FUNCTION_BLOCK INTEGRAL (* determines approximately the integral over time. *)
  (* Standard: 61499-1; Description: Copyright (c) 2024 HR Agrartechnik GmbH This program and the accompanying materials are made available under the terms of the Eclipse Public License 2.0 which is available at https://www.eclipse.org/legal/epl-2.0/ SPDX-License-Identifier: EPL-2.0 This Block was inspired by https://content.helpme-codesys.com/en/libs/Util/Current/Mathematical-Functions/INTEGRAL.html *)
  (* Version 1.0, 2024-10-18, Franz Höpfinger, HR Agrartechnik GmbH, initial Version *)
  PACKAGE utils::math;
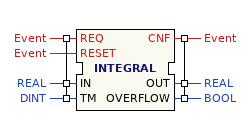
  EVENT_INPUT
    REQ WITH IN, TM; (* Normal Execution Request *)
    RESET; (* TRUE: OUT is set to zero and OVERFLOW to FALSE *)
  END_EVENT
  EVENT_OUTPUT
    CNF WITH OUT, OVERFLOW; (* Execution Confirmation *)
  END_EVENT
  VAR_INPUT
    IN : REAL := 0.0; (* Input value *)
    TM : DINT := 0; (* Time since last call in msec *)
  END_VAR
  VAR_OUTPUT
    OUT : REAL := 0.0; (* Value of the integral. This is done by summing all part integrals IN * TM *)
    OVERFLOW : BOOL := FALSE; (* TRUE: The value of OUT is out of range of REAL variables. he function is blocked till it is new initialised by input RESET. *)
  END_VAR
  ALGORITHM REQ IN ST:
IF NOT OVERFLOW THEN
	IF (1.0E38 - IN * DINT_TO_REAL(TM) < OUT OR -1.0E38 - IN * DINT_TO_REAL(TM) > OUT) THEN
		OVERFLOW := TRUE;
	ELSIF (TM > 0) THEN    // Time Difference since last call must be positive.
		OUT := OUT + IN * DINT_TO_REAL(TM) / 1000.0;
	END_IF;
END_IF;
  END_ALGORITHM
  ALGORITHM RESET IN ST:
OUT := 0.0;
OVERFLOW := FALSE;
  END_ALGORITHM
END_FUNCTION_BLOCK
